// TwinCAT 3 PLC project PLC_1
// ProgramVersion: 3.1.4026.26
// libraries:
//   Tc2_ModbusRTU, * (Beckhoff Automation GmbH)
//   Tc2_ModbusSrv, * (Beckhoff Automation GmbH)
//   Tc2_Standard, * (Beckhoff Automation GmbH)
//   Tc2_System, * (Beckhoff Automation GmbH)
// project tree:
//   GVLs/ FIO_IO.TcGVL, FIO_Modbus.TcGVL, M1_AUX.TcGVL
//   / PlcTask.TcTTO
//   POUs/COMM/ POU_COMM.TcPOU
//   POUs/CONTROL/ POU_CNTRL_M1.TcPOU, POU_CNTRL_M1_AUX.TcPOU
//   POUs/ MAIN.TcPOU
//   POUs/MAPPING/ POU_IN.TcPOU, POU_OUT.TcPOU
// real-time tasks:
//   TASK PlcTask: cycle T#10ms, priority 20, ADS port 350

CONFIGURATION PLC_1
    RESOURCE PLC ON TwinCAT3
        TASK PlcTask(INTERVAL := T#10ms, PRIORITY := 20);
        PROGRAM MAIN WITH PlcTask : MAIN;
    END_RESOURCE
END_CONFIGURATION

// ---- GVLs/FIO_IO.TcGVL
VAR_GLOBAL
	// INPUTS
	bMovingX : BOOL;
	bMovingZ : BOOL;
	bItemDetected : BOOL;
	bLidAtPlace : BOOL;
	bLidClamped : BOOL;
	bPosAtLimitLids : BOOL;
	bBaseAtPlace : BOOL;
	bBaseClamped : BOOL;
	bPosAtLimitBases : BOOL;
	bPartLiving : BOOL;
	bStart: BOOL;
	bReset : BOOL;
	bStop : BOOL;
	bEStop : BOOL;
	bAuto : BOOL;
	
	//OUTPUTS
	bMoveX : BOOL;
	bMoveZ : BOOL;
	bGrab : BOOL;
	bLidsConveyor : BOOL;
	bClampLid : BOOL;
	bPosRaiseLids : BOOL;
	bBasesConveyor : BOOL;
	bClampBase : BOOL;
	bPosRaiseBases : BOOL;
	bStartLight : BOOL;
	bResetLight : BOOL;
	bStopLight : BOOL;
END_VAR

// ---- GVLs/FIO_Modbus.TcGVL
VAR_GLOBAL
	FioInputs : ARRAY [0..15] OF BYTE;
	FioOutputs : ARRAY [0..15] OF BYTE;
END_VAR

// ---- GVLs/M1_AUX.TcGVL
VAR_GLOBAL
	ProcessTimers : ARRAY [0..20] OF TON;
END_VAR

// ---- POUs/MAIN.TcPOU
PROGRAM MAIN
VAR
END_VAR

POU_COMM();
POU_IN();
POU_CNTRL_M1_AUX();
POU_CNTRL_M1();
POU_OUT();

END_PROGRAM

// ---- POUs/COMM/POU_COMM.TcPOU
PROGRAM POU_COMM
VAR
	FBReadInputs : FB_MBReadInputs;
	FBWriteCoils : FB_MBWriteCoils;
	InputError : UDINT;
	OutputError : UDINT;
END_VAR

FBReadInputs (
	sIPAddr := '127.0.0.1',
	nTCPPort := 505,
	nUnitID := 255,
	nQuantity := 16,
	nMBAddr := 0,
	cbLength := SIZEOF(FioInputs),
	pDestAddr := ADR(FioInputs),
	bExecute := TRUE,
	tTimeout := T#1S,
	bBusy => ,
	bError => ,
	nErrId => InputError,
	cbRead => ,
);
FBReadInputs(bExecute := FALSE);


FBWriteCoils (
	sIPAddr := '127.0.0.1',
	nTCPPort := 505,
	nUnitID := 255,
	nQuantity := 16,
	nMBAddr := 0,
	cbLength := SIZEOF(FIOOutputs),
	pSrcAddr := ADR(FIOOutputs),
	bExecute := TRUE,
	tTimeout := T#1S,
	bBusy => ,
	bError => ,
	nErrId => OutputError,
	
);
FBWriteCoils(bExecute := FALSE);

END_PROGRAM

// ---- POUs/MAPPING/POU_IN.TcPOU
PROGRAM POU_IN
VAR
END_VAR

bMovingX := TO_BOOL(FioInputs[0].0);
bMovingZ := TO_BOOL(FioInputs[0].1);
bItemDetected := TO_BOOL(FioInputs[0].2);
bLidAtPlace := TO_BOOL(FioInputs[0].3);
bLidClamped := TO_BOOL(FioInputs[0].4);
bPosAtLimitLids := TO_BOOL(FioInputs[0].5);
bBaseAtPlace := TO_BOOL(FioInputs[0].6);
bBaseClamped := TO_BOOL(FioInputs[0].7);
bPosAtLimitBases := TO_BOOL(FioInputs[1].0);
bPartLiving := TO_BOOL(FioInputs[1].1);
bStart:= TO_BOOL(FioInputs[1].2);
bReset := TO_BOOL(FioInputs[1].3);
bStop := TO_BOOL(FioInputs[1].4);
bEStop := TO_BOOL(FioInputs[1].5);
bAuto := TO_BOOL(FioInputs[1].6);

END_PROGRAM

// ---- POUs/CONTROL/POU_CNTRL_M1_AUX.TcPOU
PROGRAM POU_CNTRL_M1_AUX
VAR
END_VAR

ProcessTimers[0] (
	IN := POU_CNTRL_M1.ActualStep = 50,
	PT := T#1S,
);

ProcessTimers[1] (
	IN := POU_CNTRL_M1.ActualStep = 70,
	PT := T#1S,
);

ProcessTimers[2] (
	IN := POU_CNTRL_M1.ActualStep = 80,
	PT := T#1S,
);

ProcessTimers[3] (
	IN := POU_CNTRL_M1.ActualStep = 100,
	PT := T#1S,
);

ProcessTimers[4] (
	IN := POU_CNTRL_M1.ActualStep = 100 AND ProcessTimers[3].Q,
	PT := T#3S,
);

ProcessTimers[5] (
	IN := POU_CNTRL_M1.ActualStep = 150,
	PT := T#0S,
);

ProcessTimers[6] (
	IN := POU_CNTRL_M1.ActualStep = 180,
	PT := T#1S,
);

ProcessTimers[7] (
	IN := POU_CNTRL_M1.ActualStep = 180 AND ProcessTimers[6].Q,
	PT := T#1S,
);

ProcessTimers[8] (
	IN := POU_CNTRL_M1.ActualStep = 190,
	PT := T#5S,
);

END_PROGRAM

// ---- POUs/CONTROL/POU_CNTRL_M1.TcPOU
PROGRAM POU_CNTRL_M1
VAR
	ActualStep : INT;
	NextStep : INT;
	FTrigLidAtPlace : F_TRig;
	FTRigBaseAtPlace : F_Trig;
	LidAtPlacePulse : BOOL;
	BaseAtPlacePulse : BOOL;
	FTrigPartLeaving : F_TRig;
	PartLeavingPulse : BOOL;
	ProcessStart : BOOL;
END_VAR

IF ActualStep <> NextStep THEN
	ActualStep := NextStep;
END_IF

IF (NOT bStop OR bReset) THEN
	NextStep := 0;
	ProcessStart := FALSE;
END_IF

IF bAuto AND bStart AND (bStop OR NOT bReset) THEN
	ProcessStart := TRUE;
END_IF

CASE ActualStep OF
	// machine stopped/reset
	0: 
		IF ActualStep = 0 AND NOT bAuto OR NOT bStart  THEN
			bClampBase := FALSE;
			bClampLid := FALSE;
			bMoveX := FALSE;
			bMoveZ := FALSE;
			bLidsConveyor := FALSE;
			bBasesConveyor := FALSE;
			bGrab := FALSE;
			bPosRaiseBases := FALSE;
		END_IF
	
		IF ProcessStart THEN
			bLidsConveyor := TRUE;
			bBasesConveyor := TRUE;
			NextStep := 20;
		END_IF
	
	//stop both conveyors
	20: 
		FTRigLidAtPlace (
			CLK := bLidAtPlace,
			Q => LidAtPlacePulse,
		);
		FTRigBaseAtPlace (
			CLK := bBaseAtPlace,
			Q => BaseAtPlacePulse,
		);
		
		IF BaseAtPlacePulse THEN
			bBasesConveyor := FALSE;
		END_IF
		
		IF LidAtPlacePulse THEN
			bLidsConveyor := FALSE;
		END_IF
		IF (NOT bLidsConveyor AND NOT bBasesConveyor) THEN
		NextStep := 50;
		END_IF
	
	// turn on clamp products 	
	50:
		IF NOT bLidAtPlace AND NOT bBaseAtPlace THEN
			bClampLid := TRUE;
			bClampBase := TRUE;
		END_IF
		
		IF bLidClamped AND bBaseClamped AND ProcessTimers[0].Q THEN
			NextStep := 70;
		ENd_IF
	
	// move z and turn on grab	
	70:	
		IF bLidClamped THEN
			bMoveZ := TRUE;
			IF bItemDetected THEN
				bGrab := TRUE;
			END_IF
		END_IF
		
		IF bMoveZ AND bGrab AND ProcessTimers[1].Q THEN
		NextStep := 80;
		END_IF
	
	// turn off z position	
	80:	
		IF bGrab AND bItemDetected THEN
				bMoveZ := FALSE;
		END_IF
		
		IF NOT bMoveZ AND ProcessTimers[2].Q THEN
			NextStep := 100;
		END_IF
	
	// move x and z positions
	100: 	
		IF (NOT bMoveX AND NOT bMovingX AND NOT bMoveZ AND NOT bMovingZ) THEN
			bMoveX := TRUE;
		END_IF
		IF NOT bMovingX AND bMoveX AND NOT bMoveZ AND ProcessTimers[3].Q THEN
			bMoveZ := TRUE;
		END_IF
		
		IF (bMoveX AND bMoveZ AND ProcessTimers[4].Q) THEN
			bClampLid := FALSE;	
			NextStep := 150;
		END_IF
	
	// 	turn off grab
	150:
		IF bMoveX AND bMoveZ THEN
			bGrab := FALSE;
		END_IF
		IF NOT bGrab AND ProcessTimers[5].Q THEN
		NextStep := 180;
		END_IF
		
	// turn off z and x position	
	180:
		bClampBase := FALSE;
		
		IF NOT bClampBase THEN
			bMoveZ := FALSE;
			IF NOT bMoveZ AND NOT bMovingZ AND ProcessTimers[6].Q THEN
				bMoveX := FALSE;
			END_IF	
		END_IF
		IF NOT bMoveZ AND NOT bMoveX AND NOT ProcessTimers[7].Q THEN
		NextStep := 190;
		END_IF
	
	// Raise base positioner, turn on base conveyor, wait for sensor and turn off base positioner 
	190:
		bPosRaiseBases := TRUE;
		FTrigPartLeaving (
			CLK := bPartLiving,
			Q => PartLeavingPulse,
		);
		
		IF bPosRaiseBases AND bPosAtLimitBases THEN
			bBasesConveyor := TRUE;
		END_IF
		
		IF bBasesConveyor AND PartLeavingPulse THEN
			bPosRaiseBases := FALSE;
		END_IF
		
		IF (bBasesConveyor AND NOT bPosRaiseBases AND bPosAtLimitBases) THEN
			NextStep := 200;
		END_IF
		
	// waits all conditions met and start machine again	
	200:
		IF (NOT bClampBase AND NOT bClampLid AND NOT bMoveX AND NOT bMovingX AND NOT bMoveZ AND NOT bMovingZ) THEN
 				NextStep := 0;
		END_IF
END_CASE

END_PROGRAM

// ---- POUs/MAPPING/POU_OUT.TcPOU
PROGRAM POU_OUT
VAR
END_VAR

FioOutputs[0].0 := TO_BIT(bMoveX);
FioOutputs[0].1 := TO_BIT(bMoveZ);
FioOutputs[0].2 := TO_BIT(bGrab);
FioOutputs[0].3 := TO_BIT(bLidsConveyor);
FioOutputs[0].4 := TO_BIT(bClampLid);
FioOutputs[0].5 := TO_BIT(bPosRaiseLids);
FioOutputs[0].6 := TO_BIT(bBasesConveyor);
FioOutputs[0].7 := TO_BIT(bClampBase);
FioOutputs[1].0 := TO_BIT(bPosRaiseBases);
FioOutputs[1].1 := TO_BIT(bStartLight);
FioOutputs[1].2 := TO_BIT(bResetLight);
FioOutputs[1].3 := TO_BIT(bStopLight);

END_PROGRAM
